PROGRAM MAIN
VAR
	_ivana	: BOOL;
END_VAR

END_PROGRAM

(* stored: Version 1.1.0.1, ProductVersion 3.1.4024.12
   POU MAIN: Id {a1f88fa2-3884-4087-8981-7034ef1384e1}, SpecialFunc None *)
